// TIA Portal V21 export
VAR_GLOBAL   // PLC tag table "K_SegnaliMacchina"
END_VAR
